PROGRAM PRG_04_AirValveAnalytics
VAR	
	AirValve							: ARRAY [1..6] OF Valve2Cmd2FB;
	AirValvePublishExtendMqtt			: ARRAY [1..6] OF PublishJsonMqtt;
	AirValvePublishRetractMqtt			: ARRAY [1..6] OF PublishJsonMqtt;
END_VAR


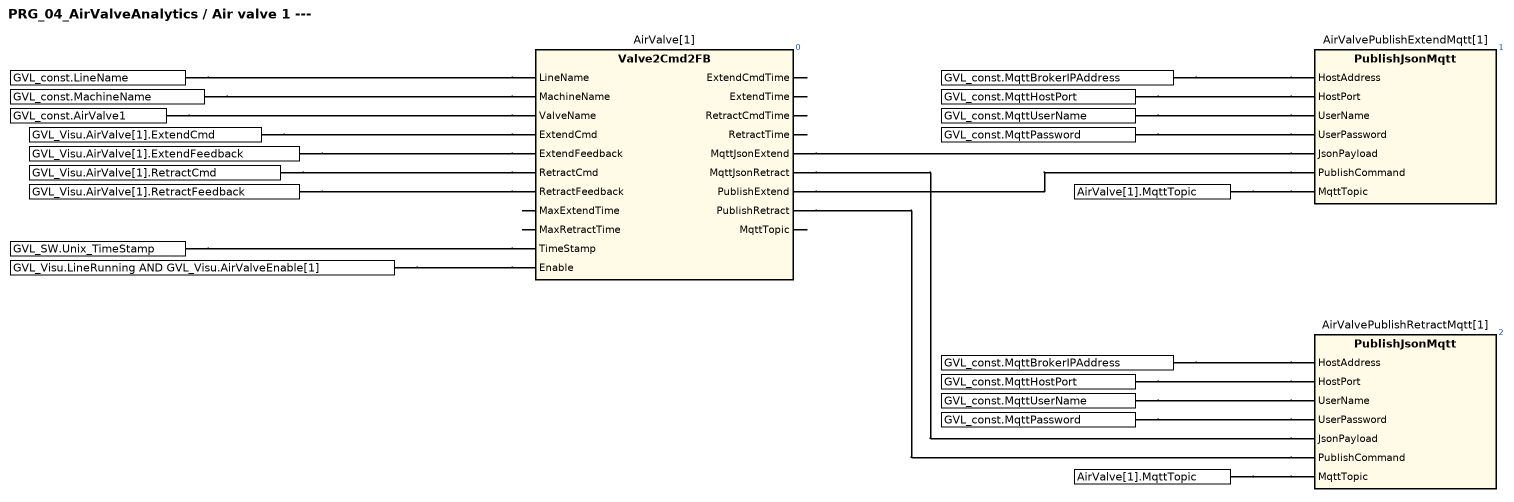
// PAGE Air valve 1 ---
AirValve[1](
    LineName := GVL_const.LineName,
    MachineName := GVL_const.MachineName,
    ValveName := GVL_const.AirValve1,
    ExtendCmd := GVL_Visu.AirValve[1].ExtendCmd,
    ExtendFeedback := GVL_Visu.AirValve[1].ExtendFeedback,
    RetractCmd := GVL_Visu.AirValve[1].RetractCmd,
    RetractFeedback := GVL_Visu.AirValve[1].RetractFeedback,
    TimeStamp := GVL_SW.Unix_TimeStamp,
    Enable := GVL_Visu.LineRunning AND GVL_Visu.AirValveEnable[1]); // Valve2Cmd2FB
AirValvePublishExtendMqtt[1](
    HostAddress := GVL_const.MqttBrokerIPAddress,
    HostPort := GVL_const.MqttHostPort,
    UserName := GVL_const.MqttUserName,
    UserPassword := GVL_const.MqttPassword,
    JsonPayload := AirValve[1].MqttJsonExtend,
    PublishCommand := AirValve[1].PublishExtend,
    MqttTopic := AirValve[1].MqttTopic); // PublishJsonMqtt
AirValvePublishRetractMqtt[1](
    HostAddress := GVL_const.MqttBrokerIPAddress,
    HostPort := GVL_const.MqttHostPort,
    UserName := GVL_const.MqttUserName,
    UserPassword := GVL_const.MqttPassword,
    JsonPayload := AirValve[1].MqttJsonRetract,
    PublishCommand := AirValve[1].PublishRetract,
    MqttTopic := AirValve[1].MqttTopic); // PublishJsonMqtt

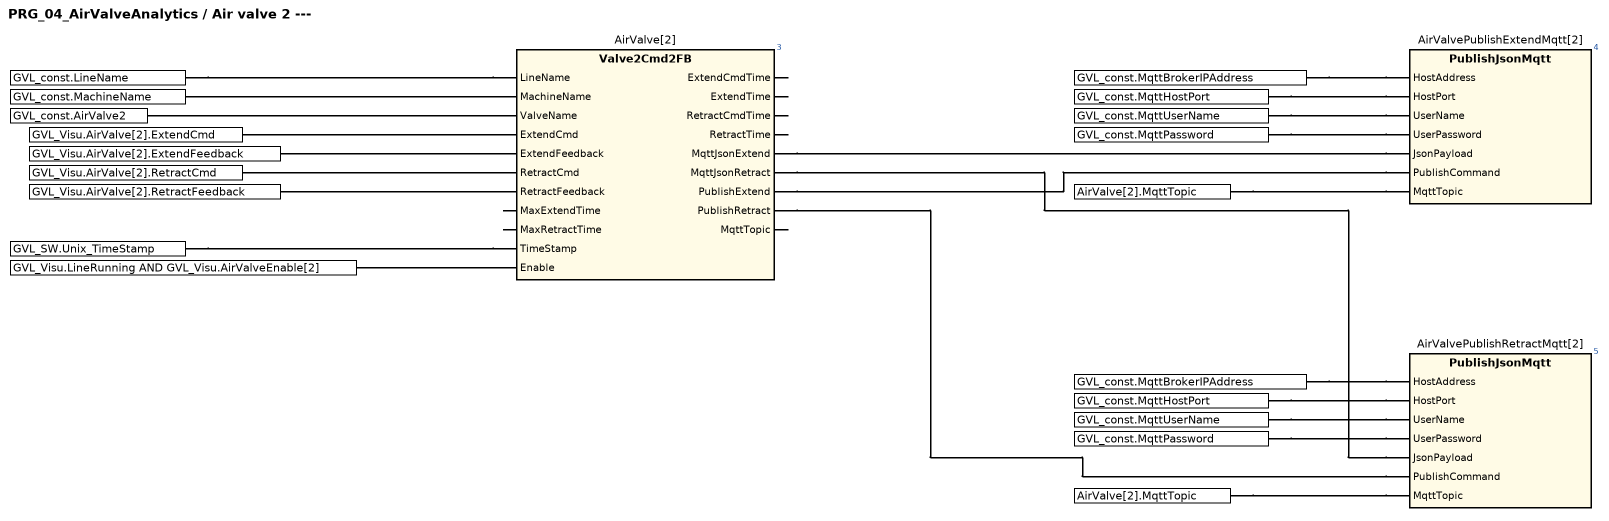
// PAGE Air valve 2 ---
AirValve[2](
    LineName := GVL_const.LineName,
    MachineName := GVL_const.MachineName,
    ValveName := GVL_const.AirValve2,
    ExtendCmd := GVL_Visu.AirValve[2].ExtendCmd,
    ExtendFeedback := GVL_Visu.AirValve[2].ExtendFeedback,
    RetractCmd := GVL_Visu.AirValve[2].RetractCmd,
    RetractFeedback := GVL_Visu.AirValve[2].RetractFeedback,
    TimeStamp := GVL_SW.Unix_TimeStamp,
    Enable := GVL_Visu.LineRunning AND GVL_Visu.AirValveEnable[2]); // Valve2Cmd2FB
AirValvePublishExtendMqtt[2](
    HostAddress := GVL_const.MqttBrokerIPAddress,
    HostPort := GVL_const.MqttHostPort,
    UserName := GVL_const.MqttUserName,
    UserPassword := GVL_const.MqttPassword,
    JsonPayload := AirValve[2].MqttJsonExtend,
    PublishCommand := AirValve[2].PublishExtend,
    MqttTopic := AirValve[2].MqttTopic); // PublishJsonMqtt
AirValvePublishRetractMqtt[2](
    HostAddress := GVL_const.MqttBrokerIPAddress,
    HostPort := GVL_const.MqttHostPort,
    UserName := GVL_const.MqttUserName,
    UserPassword := GVL_const.MqttPassword,
    JsonPayload := AirValve[2].MqttJsonRetract,
    PublishCommand := AirValve[2].PublishRetract,
    MqttTopic := AirValve[2].MqttTopic); // PublishJsonMqtt

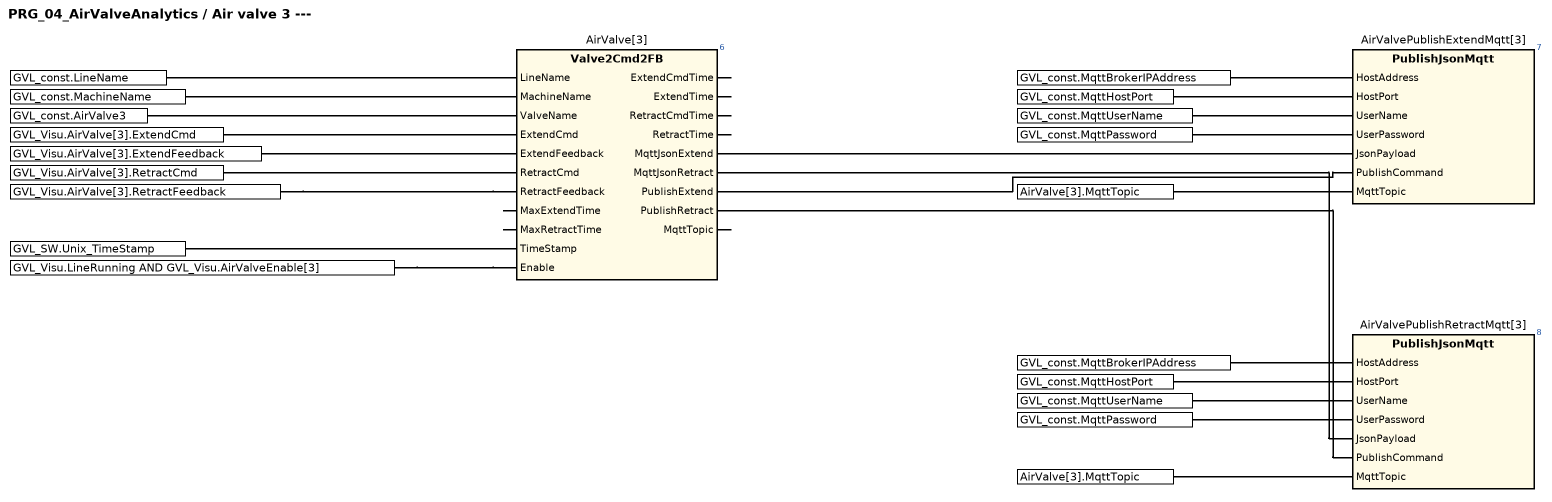
// PAGE Air valve 3 ---
AirValve[3](
    LineName := GVL_const.LineName,
    MachineName := GVL_const.MachineName,
    ValveName := GVL_const.AirValve3,
    ExtendCmd := GVL_Visu.AirValve[3].ExtendCmd,
    ExtendFeedback := GVL_Visu.AirValve[3].ExtendFeedback,
    RetractCmd := GVL_Visu.AirValve[3].RetractCmd,
    RetractFeedback := GVL_Visu.AirValve[3].RetractFeedback,
    TimeStamp := GVL_SW.Unix_TimeStamp,
    Enable := GVL_Visu.LineRunning AND GVL_Visu.AirValveEnable[3]); // Valve2Cmd2FB
AirValvePublishExtendMqtt[3](
    HostAddress := GVL_const.MqttBrokerIPAddress,
    HostPort := GVL_const.MqttHostPort,
    UserName := GVL_const.MqttUserName,
    UserPassword := GVL_const.MqttPassword,
    JsonPayload := AirValve[3].MqttJsonExtend,
    PublishCommand := AirValve[3].PublishExtend,
    MqttTopic := AirValve[3].MqttTopic); // PublishJsonMqtt
AirValvePublishRetractMqtt[3](
    HostAddress := GVL_const.MqttBrokerIPAddress,
    HostPort := GVL_const.MqttHostPort,
    UserName := GVL_const.MqttUserName,
    UserPassword := GVL_const.MqttPassword,
    JsonPayload := AirValve[3].MqttJsonRetract,
    PublishCommand := AirValve[3].PublishRetract,
    MqttTopic := AirValve[3].MqttTopic); // PublishJsonMqtt

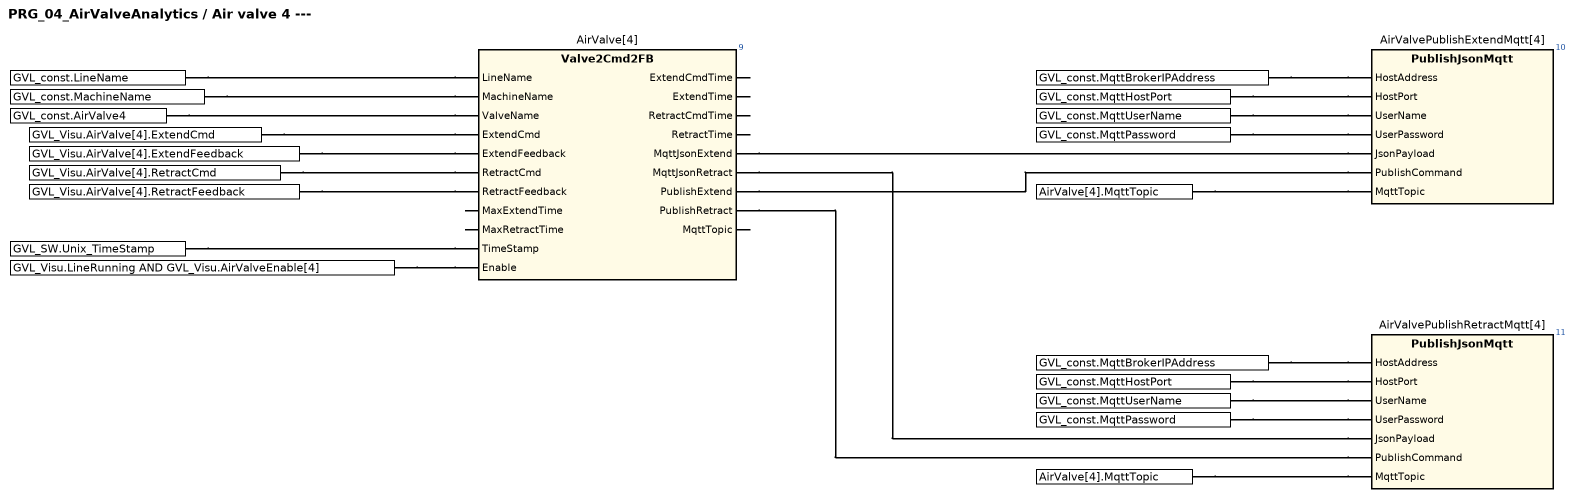
// PAGE Air valve 4 ---
AirValve[4](
    LineName := GVL_const.LineName,
    MachineName := GVL_const.MachineName,
    ValveName := GVL_const.AirValve4,
    ExtendCmd := GVL_Visu.AirValve[4].ExtendCmd,
    ExtendFeedback := GVL_Visu.AirValve[4].ExtendFeedback,
    RetractCmd := GVL_Visu.AirValve[4].RetractCmd,
    RetractFeedback := GVL_Visu.AirValve[4].RetractFeedback,
    TimeStamp := GVL_SW.Unix_TimeStamp,
    Enable := GVL_Visu.LineRunning AND GVL_Visu.AirValveEnable[4]); // Valve2Cmd2FB
AirValvePublishExtendMqtt[4](
    HostAddress := GVL_const.MqttBrokerIPAddress,
    HostPort := GVL_const.MqttHostPort,
    UserName := GVL_const.MqttUserName,
    UserPassword := GVL_const.MqttPassword,
    JsonPayload := AirValve[4].MqttJsonExtend,
    PublishCommand := AirValve[4].PublishExtend,
    MqttTopic := AirValve[4].MqttTopic); // PublishJsonMqtt
AirValvePublishRetractMqtt[4](
    HostAddress := GVL_const.MqttBrokerIPAddress,
    HostPort := GVL_const.MqttHostPort,
    UserName := GVL_const.MqttUserName,
    UserPassword := GVL_const.MqttPassword,
    JsonPayload := AirValve[4].MqttJsonRetract,
    PublishCommand := AirValve[4].PublishRetract,
    MqttTopic := AirValve[4].MqttTopic); // PublishJsonMqtt

END_PROGRAM

(* stored: Version 1.1.0.1, ProductVersion 3.1.4024.15
   POU PRG_04_AirValveAnalytics: Id {2d34a1e7-0ed3-47a9-952f-f80601f3c6db}, SpecialFunc None *)
